{attribute addProperty BoxType "EK1100-0000-0018"}
{attribute addProperty Id "Beckhoff_EM2xxxEK1122Beckhoff_EM2xxxEK1122_264CF75A162A_0001_EM2042_0000_0016EM2042_859F43D214518.125A_0002_EM2042_0000_0017EM2042_859F43D214518.125"}
{attribute addProperty CRC "3637335126"}
{attribute addProperty SizeInBites "306"}
{attribute addProperty SizeInBytes "38.25"}
TYPE Beckhoff_EM2xxx_D8CD5456 EXTENDS EK1100_179A0949 :
STRUCT
	{attribute addProperty Name "Beckhoff_EM2xxxEK1122"}
	Beckhoff_EM2xxxEK1122 : Beckhoff_EM2xxxEK1122_264CF75A;
	{attribute addProperty Name "A_0001_EM2042_0000_0016"}
	A_0001_EM2042_0000_0016 : EM2042_859F43D2;
	{attribute addProperty Name "A_0002_EM2042_0000_0017"}
	A_0002_EM2042_0000_0017 : EM2042_859F43D2;
END_STRUCT
END_TYPE

(* stored: Version 1.2.0.0, ProductVersion 3.1.4024.9
   DUT Beckhoff_EM2xxx_D8CD5456: Id {b65f8785-3afb-4d9b-8376-c2d8fe043861} *)
